Staubli VAL3: onEditItem.pgx

public program onEditItem(string& x_sEvent[], num x_nIndex, num x_nIndexItem)
  local bool l_bReachable
  local num i
  local trsf l_tApproach[2]
  local trsf l_tDepart[2]
  local num l_nSpeed
  local string l_sMessage
  local num l_nOffset
  local string l_sMessage2
  local string l_sItem
begin
  // edit the custom element that was add in the list
  if x_nIndex<6
    // edit the TRSF
    call onEditTrsf(x_nIndex,x_nIndexItem,x_sEvent)
  else
    // i=find(x_sEvent,">")+1
    call use:findPos(x_sEvent,">",i)
    i=i+1
    call language2:message(l_sMessage2,42)
    //
    switch x_nIndex
      case 6
        // change the approach 1
        call language2:message(l_sMessage,3)
        call use:changeTrsf(pEditPoint.trAppro,l_sMessage+" [1]",l_sMessage2)
      break
      case 7
        // change the approach 2
        call language2:message(l_sMessage,3)
        call use:changeTrsf(pEditPoint.trAppro[1],l_sMessage+" [2]",l_sMessage2)
      break
      case 8
        // change the approach speed
        call use:listcursor(use:nView,false)
        l_sItem=""
        call use:changeValue(pEditPoint.nSpeedApproach,1,2000,i+40-use:nBottomX,use:nView+1,l_sItem)
      break
      case 9
        // change the depart
        call language2:message(l_sMessage,4)
        call use:changeTrsf(pEditPoint.trDepart,l_sMessage+" [1]",l_sMessage2)
      break
      case 10
        // change the depart 2
        call language2:message(l_sMessage,4)
        call use:changeTrsf(pEditPoint.trDepart[1],l_sMessage+" [2]",l_sMessage2)
      break
      case 11
        // change the depart speed
        call use:listcursor(use:nView,false)
        l_sItem=""
        call use:changeValue(pEditPoint.nSpeedDepart,1,2000,i+40-use:nBottomX,use:nView+1,l_sItem)
      break
    endSwitch
  endIf
  //
end
